# EPICS autosave request: soft_iocs/galil_DMC/iocBoot/iocgalil_DMC_E06_08/all_kinematics.req
# Each DMC settings, one line per DMC
file "DMC_Kinematics.req" P=$(P1)
file "DMC_Kinematics.req" P=$(P2)
file "DMC_Kinematics.req" P=$(P3)
